// TIA Portal V16 export
// export: Created 2021-07-12T14:47:17.7050481Z, ExportSetting WithDefaults, DisplayName Totally Integrated Automation Portal, DisplayVersion V16, DisplayName TIA Portal Version Control Interface, DisplayVersion V16, DisplayName TIA Portal Openness, DisplayVersion V16, DisplayName STEP 7 Professional, DisplayVersion V16, DisplayName STEP 7 Safety, DisplayVersion V16, DisplayName WinCC Professional, DisplayVersion V16
TYPE "LSimaHydTO_typeMeasurementQOutputRange"
TITLE = LSimaHydTO_typeMeasurementQOutputRange
// stored: IsFailsafeCompliant false
   STRUCT
      maxQOutputValue { S7_SetPoint := 'True'} : Real;   // incremented up to this value
      numberOfPoints { S7_SetPoint := 'True'} : Int;   // number of points for this range
   END_STRUCT;
END_TYPE
